// TwinCAT 3 PLC project Plc
// ProgramVersion: 3.1.4023.0
// libraries:
//   Tc2_Standard, * (Beckhoff Automation GmbH)
//   Tc2_System, * (Beckhoff Automation GmbH)
//   Tc3_Module, * (Beckhoff Automation GmbH)
// project tree:
//   / PlcTask.TcTTO (not stored)
//   DUTs/IO/PdoEntries/ FSOE_31BB7F2A.TcDUT, FSOE_3C294B21.TcDUT, FSOE_13BCEA3F.TcDUT, FSOE_6A82EB93.TcDUT, FSOE_BB3344D6.TcDUT
//   DUTs/IO/PDOs/ DeviceMain_Outputs_650F3486.TcDUT, FSoE_Slave_Connection_1_Slave_Message_330A35E4.TcDUT, Standard_Inputdata_FDD1436A.TcDUT, FSLOGIC_Inputs_CD3F9A93.TcDUT, FSoE_Slave_Connection_1_Master_Message_7109E4F0.TcDUT, Standard_Outputdata_59C030BE.TcDUT, EMPTY_STRUCTURE.TcDUT, Ch_A_AxisMain_Inputs_BA7CE8DB.TcDUT, Ch_A_AxisMain_Outputs_A99AE12E.TcDUT, Ch_A_Interpolator_Outputs_462A5F1D.TcDUT, Ch_A_PositionControl_Inputs_8CB0F55A.TcDUT, WcState_B516A264.TcDUT, InfoData_358A59CF.TcDUT, Device_6E257577.TcDUT, Device_Safety_C21945A1.TcDUT, Ch_A_D18C6F16.TcDUT, InfoData_E68C61CD.TcDUT (not stored), WcState_0B2B16F9.TcDUT (not stored), InfoData_2A97D6CF.TcDUT (not stored), Inputs_A65FACA4.TcDUT (not stored), Outputs_23C0ED1D.TcDUT (not stored)
//   DUTs/IO/Boxes/ AMP8000_F7A82895.TcDUT
//   DUTs/IO/Devices/ SyncUnitTask_2D604ED5.TcDUT (not stored), SyncUnitTasks_6FEB8257.TcDUT (not stored), SyncUnits_99E584AF.TcDUT (not stored)
//   DUTs/IO/Topology/ Device_1_EtherCAT_60A1425B.TcDUT (not stored)
//   DUTs/IO/Base/ EtcSlaveBase_82538BE2.TcDUT (not stored), EtcSlaveBase_82538BE2.TcDUT (not stored), EtcSlaveBase_82538BE2.TcDUT (not stored), EtcSlaveTerminalBase_947E5A46.TcDUT (not stored), EtcSlaveBoxBase_77A0E4A7.TcDUT (not stored), EtcSlaveEndTerminalBase_866C7F0C.TcDUT (not stored), InputBase_8311D824.TcDUT (not stored), OutputBase_10CEE7DE.TcDUT (not stored), EtcMasterBase_62654B43.TcDUT (not stored)
//   GVLs/ GVL_iXlinker.TcGVL (not stored)
// real-time tasks:
//   TASK PlcTask: cycle T#10ms, priority 20, ADS port 350
// I/O:
//   DEVICE Device 1 (EtherCAT), AmsNetId 172.20.30.238.2.1
//     Drive 1 (AMP8000-0030-0103) [AMP8000-0030-0103]
//       modules: Device, Device, Device, Device, Device, Device, Device, Device, Device, Device, Device (Safety), Device, Device, Device, Device, Device, Device, Device, Device, Device, Device, Device, Device, Device, Device, Device, Device, Device, Device, Device, Device, Ch A, Ch A, Ch A, Ch A, Ch A, Ch A, Ch A, Ch A, Ch A, Ch A, Ch A, Ch A, Ch A, Ch A, Ch A, Ch A, Ch A, Ch A, Ch A, Ch A, Ch A, Ch A, Ch A, Ch A, Ch A, Ch A
// variable links:
//   Plc/Plc Instance <-> Device 1 (EtherCAT)/Drive 1 (AMP8000-0030-0103)
//     PlcTask Outputs/GVL_iXlinker.Device_1_EtherCAT.Drive_1_AMP8000_0030_0103.Device.DeviceMain_Outputs.Power_supply_controlword <-> Device/DeviceMain Outputs/Power supply controlword
//     PlcTask Inputs/GVL_iXlinker.Device_1_EtherCAT.Drive_1_AMP8000_0030_0103.Device_Safety.FSoE_Slave_Connection_1_Slave_Message.FSOE/FSoE_Slave_Cmd <-> Device (Safety)/FSoE Slave Connection 1 Slave Message/FSOE/FSoE Slave Cmd
//     PlcTask Inputs/GVL_iXlinker.Device_1_EtherCAT.Drive_1_AMP8000_0030_0103.Device_Safety.FSoE_Slave_Connection_1_Slave_Message.FSOE/Axis_A_STO <-> Device (Safety)/FSoE Slave Connection 1 Slave Message/FSOE/Axis A STO
//     PlcTask Inputs/GVL_iXlinker.Device_1_EtherCAT.Drive_1_AMP8000_0030_0103.Device_Safety.FSoE_Slave_Connection_1_Slave_Message.FSOE/Safe_Input_1 <-> Device (Safety)/FSoE Slave Connection 1 Slave Message/FSOE/Safe Input_1
//     PlcTask Inputs/GVL_iXlinker.Device_1_EtherCAT.Drive_1_AMP8000_0030_0103.Device_Safety.FSoE_Slave_Connection_1_Slave_Message.FSOE/Safe_Input_2 <-> Device (Safety)/FSoE Slave Connection 1 Slave Message/FSOE/Safe Input_2
//     PlcTask Inputs/GVL_iXlinker.Device_1_EtherCAT.Drive_1_AMP8000_0030_0103.Device_Safety.FSoE_Slave_Connection_1_Slave_Message.FSOE/Safe_Input_3 <-> Device (Safety)/FSoE Slave Connection 1 Slave Message/FSOE/Safe Input_3
//     PlcTask Inputs/GVL_iXlinker.Device_1_EtherCAT.Drive_1_AMP8000_0030_0103.Device_Safety.FSoE_Slave_Connection_1_Slave_Message.FSOE/Safe_Input_4 <-> Device (Safety)/FSoE Slave Connection 1 Slave Message/FSOE/Safe Input_4
//     PlcTask Inputs/GVL_iXlinker.Device_1_EtherCAT.Drive_1_AMP8000_0030_0103.Device_Safety.FSoE_Slave_Connection_1_Slave_Message.FSOE/Safe_Input_5 <-> Device (Safety)/FSoE Slave Connection 1 Slave Message/FSOE/Safe Input_5
//     PlcTask Inputs/GVL_iXlinker.Device_1_EtherCAT.Drive_1_AMP8000_0030_0103.Device_Safety.FSoE_Slave_Connection_1_Slave_Message.FSOE/Safe_Input_6 <-> Device (Safety)/FSoE Slave Connection 1 Slave Message/FSOE/Safe Input_6
//     PlcTask Inputs/GVL_iXlinker.Device_1_EtherCAT.Drive_1_AMP8000_0030_0103.Device_Safety.FSoE_Slave_Connection_1_Slave_Message.FSOE/Safe_Input_7 <-> Device (Safety)/FSoE Slave Connection 1 Slave Message/FSOE/Safe Input_7
//     PlcTask Inputs/GVL_iXlinker.Device_1_EtherCAT.Drive_1_AMP8000_0030_0103.Device_Safety.FSoE_Slave_Connection_1_Slave_Message.FSOE/Safe_Input_9 <-> Device (Safety)/FSoE Slave Connection 1 Slave Message/FSOE/Safe Input_9
//     PlcTask Inputs/GVL_iXlinker.Device_1_EtherCAT.Drive_1_AMP8000_0030_0103.Device_Safety.FSoE_Slave_Connection_1_Slave_Message.FSOE/Safe_Input_10 <-> Device (Safety)/FSoE Slave Connection 1 Slave Message/FSOE/Safe Input_10
//     PlcTask Inputs/GVL_iXlinker.Device_1_EtherCAT.Drive_1_AMP8000_0030_0103.Device_Safety.FSoE_Slave_Connection_1_Slave_Message.FSOE/Safe_Input_11 <-> Device (Safety)/FSoE Slave Connection 1 Slave Message/FSOE/Safe Input_11
//     PlcTask Inputs/GVL_iXlinker.Device_1_EtherCAT.Drive_1_AMP8000_0030_0103.Device_Safety.FSoE_Slave_Connection_1_Slave_Message.FSOE/Safe_Input_12 <-> Device (Safety)/FSoE Slave Connection 1 Slave Message/FSOE/Safe Input_12
//     PlcTask Inputs/GVL_iXlinker.Device_1_EtherCAT.Drive_1_AMP8000_0030_0103.Device_Safety.FSoE_Slave_Connection_1_Slave_Message.FSOE/Safe_Input_13 <-> Device (Safety)/FSoE Slave Connection 1 Slave Message/FSOE/Safe Input_13
//     PlcTask Inputs/GVL_iXlinker.Device_1_EtherCAT.Drive_1_AMP8000_0030_0103.Device_Safety.FSoE_Slave_Connection_1_Slave_Message.FSOE/Safe_Input_14 <-> Device (Safety)/FSoE Slave Connection 1 Slave Message/FSOE/Safe Input_14
//     PlcTask Inputs/GVL_iXlinker.Device_1_EtherCAT.Drive_1_AMP8000_0030_0103.Device_Safety.FSoE_Slave_Connection_1_Slave_Message.FSOE/Safe_Input_15 <-> Device (Safety)/FSoE Slave Connection 1 Slave Message/FSOE/Safe Input_15
//     PlcTask Inputs/GVL_iXlinker.Device_1_EtherCAT.Drive_1_AMP8000_0030_0103.Device_Safety.FSoE_Slave_Connection_1_Slave_Message.FSOE/Axis_B_STO <-> Device (Safety)/FSoE Slave Connection 1 Slave Message/FSOE/Axis B STO
//     PlcTask Inputs/GVL_iXlinker.Device_1_EtherCAT.Drive_1_AMP8000_0030_0103.Device_Safety.FSoE_Slave_Connection_1_Slave_Message.FSOE/FSoE_Slave_CRC_0 <-> Device (Safety)/FSoE Slave Connection 1 Slave Message/FSOE/FSoE Slave CRC_0
//     PlcTask Inputs/GVL_iXlinker.Device_1_EtherCAT.Drive_1_AMP8000_0030_0103.Device_Safety.FSoE_Slave_Connection_1_Slave_Message.FSOE/FSoE_Slave_ConnID <-> Device (Safety)/FSoE Slave Connection 1 Slave Message/FSOE/FSoE Slave ConnID
//     PlcTask Inputs/GVL_iXlinker.Device_1_EtherCAT.Drive_1_AMP8000_0030_0103.Device_Safety.Standard_Inputdata.FSOE/Std_Input <-> Device (Safety)/Standard Inputdata/FSOE/Std Input
//     PlcTask Inputs/GVL_iXlinker.Device_1_EtherCAT.Drive_1_AMP8000_0030_0103.Device_Safety.Standard_Inputdata.FSOE/Std_Input_1 <-> Device (Safety)/Standard Inputdata/FSOE/Std Input_1
//     PlcTask Inputs/GVL_iXlinker.Device_1_EtherCAT.Drive_1_AMP8000_0030_0103.Device_Safety.Standard_Inputdata.FSOE/Std_Input_2 <-> Device (Safety)/Standard Inputdata/FSOE/Std Input_2
//     PlcTask Inputs/GVL_iXlinker.Device_1_EtherCAT.Drive_1_AMP8000_0030_0103.Device_Safety.Standard_Inputdata.FSOE/Std_Input_3 <-> Device (Safety)/Standard Inputdata/FSOE/Std Input_3
//     PlcTask Inputs/GVL_iXlinker.Device_1_EtherCAT.Drive_1_AMP8000_0030_0103.Device_Safety.Standard_Inputdata.FSOE/Std_Input_4 <-> Device (Safety)/Standard Inputdata/FSOE/Std Input_4
//     PlcTask Inputs/GVL_iXlinker.Device_1_EtherCAT.Drive_1_AMP8000_0030_0103.Device_Safety.Standard_Inputdata.FSOE/Std_Input_5 <-> Device (Safety)/Standard Inputdata/FSOE/Std Input_5
//     PlcTask Inputs/GVL_iXlinker.Device_1_EtherCAT.Drive_1_AMP8000_0030_0103.Device_Safety.Standard_Inputdata.FSOE/Std_Input_6 <-> Device (Safety)/Standard Inputdata/FSOE/Std Input_6
//     PlcTask Inputs/GVL_iXlinker.Device_1_EtherCAT.Drive_1_AMP8000_0030_0103.Device_Safety.Standard_Inputdata.FSOE/Std_Input_7 <-> Device (Safety)/Standard Inputdata/FSOE/Std Input_7
//     PlcTask Inputs/GVL_iXlinker.Device_1_EtherCAT.Drive_1_AMP8000_0030_0103.Device_Safety.FSLOGIC_Inputs.FSOE/Safe_Logic_State <-> Device (Safety)/FSLOGIC Inputs/FSOE/Safe Logic State
//     PlcTask Inputs/GVL_iXlinker.Device_1_EtherCAT.Drive_1_AMP8000_0030_0103.Device_Safety.FSLOGIC_Inputs.FSOE/Cycle_Counter <-> Device (Safety)/FSLOGIC Inputs/FSOE/Cycle Counter
//     PlcTask Outputs/GVL_iXlinker.Device_1_EtherCAT.Drive_1_AMP8000_0030_0103.Device_Safety.FSoE_Slave_Connection_1_Master_Message.FSOE/FSoE_Master_Cmd <-> Device (Safety)/FSoE Slave Connection 1 Master Message/FSOE/FSoE Master Cmd
//     PlcTask Outputs/GVL_iXlinker.Device_1_EtherCAT.Drive_1_AMP8000_0030_0103.Device_Safety.FSoE_Slave_Connection_1_Master_Message.FSOE/Axis_A_STO <-> Device (Safety)/FSoE Slave Connection 1 Master Message/FSOE/Axis A STO
//     PlcTask Outputs/GVL_iXlinker.Device_1_EtherCAT.Drive_1_AMP8000_0030_0103.Device_Safety.FSoE_Slave_Connection_1_Master_Message.FSOE/Safe_Output_1 <-> Device (Safety)/FSoE Slave Connection 1 Master Message/FSOE/Safe Output_1
//     PlcTask Outputs/GVL_iXlinker.Device_1_EtherCAT.Drive_1_AMP8000_0030_0103.Device_Safety.FSoE_Slave_Connection_1_Master_Message.FSOE/Safe_Output_2 <-> Device (Safety)/FSoE Slave Connection 1 Master Message/FSOE/Safe Output_2
//     PlcTask Outputs/GVL_iXlinker.Device_1_EtherCAT.Drive_1_AMP8000_0030_0103.Device_Safety.FSoE_Slave_Connection_1_Master_Message.FSOE/Safe_Output_3 <-> Device (Safety)/FSoE Slave Connection 1 Master Message/FSOE/Safe Output_3
//     PlcTask Outputs/GVL_iXlinker.Device_1_EtherCAT.Drive_1_AMP8000_0030_0103.Device_Safety.FSoE_Slave_Connection_1_Master_Message.FSOE/Safe_Output_4 <-> Device (Safety)/FSoE Slave Connection 1 Master Message/FSOE/Safe Output_4
//     PlcTask Outputs/GVL_iXlinker.Device_1_EtherCAT.Drive_1_AMP8000_0030_0103.Device_Safety.FSoE_Slave_Connection_1_Master_Message.FSOE/Safe_Output_5 <-> Device (Safety)/FSoE Slave Connection 1 Master Message/FSOE/Safe Output_5
//     PlcTask Outputs/GVL_iXlinker.Device_1_EtherCAT.Drive_1_AMP8000_0030_0103.Device_Safety.FSoE_Slave_Connection_1_Master_Message.FSOE/Safe_Output_6 <-> Device (Safety)/FSoE Slave Connection 1 Master Message/FSOE/Safe Output_6
//     PlcTask Outputs/GVL_iXlinker.Device_1_EtherCAT.Drive_1_AMP8000_0030_0103.Device_Safety.FSoE_Slave_Connection_1_Master_Message.FSOE/Safe_Output_7 <-> Device (Safety)/FSoE Slave Connection 1 Master Message/FSOE/Safe Output_7
//     PlcTask Outputs/GVL_iXlinker.Device_1_EtherCAT.Drive_1_AMP8000_0030_0103.Device_Safety.FSoE_Slave_Connection_1_Master_Message.FSOE/Safe_Output_9 <-> Device (Safety)/FSoE Slave Connection 1 Master Message/FSOE/Safe Output_9
//     PlcTask Outputs/GVL_iXlinker.Device_1_EtherCAT.Drive_1_AMP8000_0030_0103.Device_Safety.FSoE_Slave_Connection_1_Master_Message.FSOE/Safe_Output_10 <-> Device (Safety)/FSoE Slave Connection 1 Master Message/FSOE/Safe Output_10
//     PlcTask Outputs/GVL_iXlinker.Device_1_EtherCAT.Drive_1_AMP8000_0030_0103.Device_Safety.FSoE_Slave_Connection_1_Master_Message.FSOE/Safe_Output_11 <-> Device (Safety)/FSoE Slave Connection 1 Master Message/FSOE/Safe Output_11
//     PlcTask Outputs/GVL_iXlinker.Device_1_EtherCAT.Drive_1_AMP8000_0030_0103.Device_Safety.FSoE_Slave_Connection_1_Master_Message.FSOE/Safe_Output_12 <-> Device (Safety)/FSoE Slave Connection 1 Master Message/FSOE/Safe Output_12
//     PlcTask Outputs/GVL_iXlinker.Device_1_EtherCAT.Drive_1_AMP8000_0030_0103.Device_Safety.FSoE_Slave_Connection_1_Master_Message.FSOE/Safe_Output_13 <-> Device (Safety)/FSoE Slave Connection 1 Master Message/FSOE/Safe Output_13
//     PlcTask Outputs/GVL_iXlinker.Device_1_EtherCAT.Drive_1_AMP8000_0030_0103.Device_Safety.FSoE_Slave_Connection_1_Master_Message.FSOE/Safe_Output_14 <-> Device (Safety)/FSoE Slave Connection 1 Master Message/FSOE/Safe Output_14
//     PlcTask Outputs/GVL_iXlinker.Device_1_EtherCAT.Drive_1_AMP8000_0030_0103.Device_Safety.FSoE_Slave_Connection_1_Master_Message.FSOE/Safe_Output_15 <-> Device (Safety)/FSoE Slave Connection 1 Master Message/FSOE/Safe Output_15
//     PlcTask Outputs/GVL_iXlinker.Device_1_EtherCAT.Drive_1_AMP8000_0030_0103.Device_Safety.FSoE_Slave_Connection_1_Master_Message.FSOE/Axis_B_STO <-> Device (Safety)/FSoE Slave Connection 1 Master Message/FSOE/Axis B STO
//     PlcTask Outputs/GVL_iXlinker.Device_1_EtherCAT.Drive_1_AMP8000_0030_0103.Device_Safety.FSoE_Slave_Connection_1_Master_Message.FSOE/FSoE_Master_CRC_0 <-> Device (Safety)/FSoE Slave Connection 1 Master Message/FSOE/FSoE Master CRC_0
//     PlcTask Outputs/GVL_iXlinker.Device_1_EtherCAT.Drive_1_AMP8000_0030_0103.Device_Safety.FSoE_Slave_Connection_1_Master_Message.FSOE/FSoE_Master_ConnID <-> Device (Safety)/FSoE Slave Connection 1 Master Message/FSOE/FSoE Master ConnID
//     PlcTask Outputs/GVL_iXlinker.Device_1_EtherCAT.Drive_1_AMP8000_0030_0103.Device_Safety.Standard_Outputdata.FSOE/Std_Output <-> Device (Safety)/Standard Outputdata/FSOE/Std Output
//     PlcTask Outputs/GVL_iXlinker.Device_1_EtherCAT.Drive_1_AMP8000_0030_0103.Device_Safety.Standard_Outputdata.FSOE/Std_Output_1 <-> Device (Safety)/Standard Outputdata/FSOE/Std Output_1
//     PlcTask Outputs/GVL_iXlinker.Device_1_EtherCAT.Drive_1_AMP8000_0030_0103.Device_Safety.Standard_Outputdata.FSOE/Std_Output_2 <-> Device (Safety)/Standard Outputdata/FSOE/Std Output_2
//     PlcTask Outputs/GVL_iXlinker.Device_1_EtherCAT.Drive_1_AMP8000_0030_0103.Device_Safety.Standard_Outputdata.FSOE/Std_Output_3 <-> Device (Safety)/Standard Outputdata/FSOE/Std Output_3
//     PlcTask Outputs/GVL_iXlinker.Device_1_EtherCAT.Drive_1_AMP8000_0030_0103.Device_Safety.Standard_Outputdata.FSOE/Std_Output_4 <-> Device (Safety)/Standard Outputdata/FSOE/Std Output_4
//     PlcTask Outputs/GVL_iXlinker.Device_1_EtherCAT.Drive_1_AMP8000_0030_0103.Device_Safety.Standard_Outputdata.FSOE/Std_Output_5 <-> Device (Safety)/Standard Outputdata/FSOE/Std Output_5
//     PlcTask Outputs/GVL_iXlinker.Device_1_EtherCAT.Drive_1_AMP8000_0030_0103.Device_Safety.Standard_Outputdata.FSOE/Std_Output_6 <-> Device (Safety)/Standard Outputdata/FSOE/Std Output_6
//     PlcTask Outputs/GVL_iXlinker.Device_1_EtherCAT.Drive_1_AMP8000_0030_0103.Device_Safety.Standard_Outputdata.FSOE/Std_Output_7 <-> Device (Safety)/Standard Outputdata/FSOE/Std Output_7
//     PlcTask Inputs/GVL_iXlinker.Device_1_EtherCAT.Drive_1_AMP8000_0030_0103.Ch_A.Ch_A_AxisMain_Inputs.Position_actual_value_invalid <-> Ch A/Ch A AxisMain Inputs/Position actual value invalid
//     PlcTask Inputs/GVL_iXlinker.Device_1_EtherCAT.Drive_1_AMP8000_0030_0103.Ch_A.Ch_A_AxisMain_Inputs._1st_Additional_position_actual_value_invalid <-> Ch A/Ch A AxisMain Inputs/1st Additional position actual value invalid
//     PlcTask Inputs/GVL_iXlinker.Device_1_EtherCAT.Drive_1_AMP8000_0030_0103.Ch_A.Ch_A_AxisMain_Inputs.Ch_A_Statusword <-> Ch A/Ch A AxisMain Inputs/Ch A Statusword
//     PlcTask Inputs/GVL_iXlinker.Device_1_EtherCAT.Drive_1_AMP8000_0030_0103.Ch_A.Ch_A_AxisMain_Inputs.Ch_A_Position_actual_value <-> Ch A/Ch A AxisMain Inputs/Ch A Position actual value
//     PlcTask Outputs/GVL_iXlinker.Device_1_EtherCAT.Drive_1_AMP8000_0030_0103.Ch_A.Ch_A_AxisMain_Outputs.Ch_A_Controlword <-> Ch A/Ch A AxisMain Outputs/Ch A Controlword
//     PlcTask Outputs/GVL_iXlinker.Device_1_EtherCAT.Drive_1_AMP8000_0030_0103.Ch_A.Ch_A_Interpolator_Outputs.Ch_A_Target_position <-> Ch A/Ch A Interpolator Outputs/Ch A Target position
//     PlcTask Outputs/GVL_iXlinker.Device_1_EtherCAT.Drive_1_AMP8000_0030_0103.Ch_A.Ch_A_Interpolator_Outputs.Ch_A_Target_velocity <-> Ch A/Ch A Interpolator Outputs/Ch A Target velocity
//     PlcTask Inputs/GVL_iXlinker.Device_1_EtherCAT.Drive_1_AMP8000_0030_0103.Ch_A.Ch_A_PositionControl_Inputs.Ch_A_Following_error_actual_value <-> Ch A/Ch A PositionControl Inputs/Ch A Following error actual value
//     PlcTask Inputs/GVL_iXlinker.Device_1_EtherCAT.Drive_1_AMP8000_0030_0103.WcState.WcState0 <-> WcState/WcState0
//     PlcTask Inputs/GVL_iXlinker.Device_1_EtherCAT.Drive_1_AMP8000_0030_0103.WcState.WcState1 <-> WcState/WcState1
//     PlcTask Inputs/GVL_iXlinker.Device_1_EtherCAT.Drive_1_AMP8000_0030_0103.WcState.InputToggle0 <-> WcState/InputToggle0
//     PlcTask Inputs/GVL_iXlinker.Device_1_EtherCAT.Drive_1_AMP8000_0030_0103.WcState.InputToggle1 <-> WcState/InputToggle1
//     PlcTask Inputs/GVL_iXlinker.Device_1_EtherCAT.Drive_1_AMP8000_0030_0103.InfoData.AdsAddr <-> InfoData/AdsAddr
//     PlcTask Inputs/GVL_iXlinker.Device_1_EtherCAT.Drive_1_AMP8000_0030_0103.InfoData.DcOutputShift <-> InfoData/DcOutputShift
//     PlcTask Inputs/GVL_iXlinker.Device_1_EtherCAT.Drive_1_AMP8000_0030_0103.InfoData.DcInputShift <-> InfoData/DcInputShift
//     PlcTask Inputs/GVL_iXlinker.Device_1_EtherCAT.Drive_1_AMP8000_0030_0103.InfoData.AoeNetId <-> InfoData/AoeNetId
//     PlcTask Inputs/GVL_iXlinker.Device_1_EtherCAT.Drive_1_AMP8000_0030_0103.InfoData.Chn0 <-> InfoData/Chn0
//     PlcTask Inputs/GVL_iXlinker.Device_1_EtherCAT.Drive_1_AMP8000_0030_0103.InfoData.State <-> InfoData/State
//   Plc/Plc Instance <-> Device 1 (EtherCAT)
//     PlcTask Inputs/GVL_iXlinker.Device_1_EtherCAT.SyncUnits._default._unreferenced.WcState.WcState <-> SyncUnits/<default>/<unreferenced>/WcState/WcState
//     PlcTask Inputs/GVL_iXlinker.Device_1_EtherCAT.SyncUnits._default._unreferenced.InfoData.ObjectId <-> SyncUnits/<default>/<unreferenced>/InfoData/ObjectId
//     PlcTask Inputs/GVL_iXlinker.Device_1_EtherCAT.SyncUnits._default._unreferenced.InfoData.State <-> SyncUnits/<default>/<unreferenced>/InfoData/State
//     PlcTask Inputs/GVL_iXlinker.Device_1_EtherCAT.SyncUnits._default._unreferenced.InfoData.SlaveCount <-> SyncUnits/<default>/<unreferenced>/InfoData/SlaveCount
//     PlcTask Inputs/GVL_iXlinker.Device_1_EtherCAT.SyncUnits._default.PlcTask.WcState.WcState <-> SyncUnits/<default>/PlcTask/WcState/WcState
//     PlcTask Inputs/GVL_iXlinker.Device_1_EtherCAT.SyncUnits._default.PlcTask.InfoData.ObjectId <-> SyncUnits/<default>/PlcTask/InfoData/ObjectId
//     PlcTask Inputs/GVL_iXlinker.Device_1_EtherCAT.SyncUnits._default.PlcTask.InfoData.State <-> SyncUnits/<default>/PlcTask/InfoData/State
//     PlcTask Inputs/GVL_iXlinker.Device_1_EtherCAT.SyncUnits._default.PlcTask.InfoData.SlaveCount <-> SyncUnits/<default>/PlcTask/InfoData/SlaveCount
//     PlcTask Inputs/GVL_iXlinker.Device_1_EtherCAT.Inputs.SlaveCount <-> Inputs/SlaveCount
//     PlcTask Inputs/GVL_iXlinker.Device_1_EtherCAT.Inputs.DevState <-> Inputs/DevState
//     PlcTask Inputs/GVL_iXlinker.Device_1_EtherCAT.Inputs.Frm0State <-> Inputs/Frm0State
//     PlcTask Inputs/GVL_iXlinker.Device_1_EtherCAT.Inputs.Frm0WcState <-> Inputs/Frm0WcState
//     PlcTask Inputs/GVL_iXlinker.Device_1_EtherCAT.Inputs.Frm0InputToggle <-> Inputs/Frm0InputToggle
//     PlcTask Outputs/GVL_iXlinker.Device_1_EtherCAT.Outputs.DevCtrl <-> Outputs/DevCtrl
//     PlcTask Outputs/GVL_iXlinker.Device_1_EtherCAT.Outputs.Frm0Ctrl <-> Outputs/Frm0Ctrl
//     PlcTask Outputs/GVL_iXlinker.Device_1_EtherCAT.Outputs.Frm0WcCtrl <-> Outputs/Frm0WcCtrl
//     PlcTask Inputs/GVL_iXlinker.Device_1_EtherCAT.InfoData.ChangeCount <-> InfoData/ChangeCount
//     PlcTask Inputs/GVL_iXlinker.Device_1_EtherCAT.InfoData.DevId <-> InfoData/DevId
//     PlcTask Inputs/GVL_iXlinker.Device_1_EtherCAT.InfoData.AmsNetId <-> InfoData/AmsNetId
//     PlcTask Inputs/GVL_iXlinker.Device_1_EtherCAT.InfoData.CfgSlaveCount <-> InfoData/CfgSlaveCount
//     PlcTask Inputs/GVL_iXlinker.Device_1_EtherCAT.InfoData.DcToTcTimeOffset <-> InfoData/DcToTcTimeOffset
//     PlcTask Inputs/GVL_iXlinker.Device_1_EtherCAT.InfoData.DcToExtTimeOffset <-> InfoData/DcToExtTimeOffset

// ---- DUTs/IO/PdoEntries/FSOE_31BB7F2A.TcDUT
{attribute 'GeneratedUsingTerminal: AMP8000-0030-0103-0103'}
{attribute addProperty BoxType "AMP8000-0030-0103-0103"}
{attribute addProperty Id "FSoE_Slave_CmdUSINT1Axis_A_STOBOOL1Safe_Input_1BOOL1Safe_Input_2BOOL1Safe_Input_3BOOL1Safe_Input_4BOOL1Safe_Input_5BOOL1Safe_Input_6BOOL1Safe_Input_7BOOL1Axis_B_STOBOOL1Safe_Input_9BOOL1Safe_Input_10BOOL1Safe_Input_11BOOL1Safe_Input_12BOOL1Safe_Input_13BOOL1Safe_Input_14BOOL1Safe_Input_15BOOL1FSoE_Slave_CRC_0UINT2FSoE_Slave_ConnIDUINT2"}
{attribute addProperty CRC "834371370"}
{attribute addProperty Size "21"}
TYPE FSOE_31BB7F2A :
STRUCT
	{attribute addProperty Name "FSoE_Slave_Cmd"}
	FSoE_Slave_Cmd : USINT;
	{attribute addProperty Name "Axis_A_STO"}
	Axis_A_STO : BOOL;
	{attribute addProperty Name "Safe_Input_1"}
	Safe_Input_1 : BOOL;
	{attribute addProperty Name "Safe_Input_2"}
	Safe_Input_2 : BOOL;
	{attribute addProperty Name "Safe_Input_3"}
	Safe_Input_3 : BOOL;
	{attribute addProperty Name "Safe_Input_4"}
	Safe_Input_4 : BOOL;
	{attribute addProperty Name "Safe_Input_5"}
	Safe_Input_5 : BOOL;
	{attribute addProperty Name "Safe_Input_6"}
	Safe_Input_6 : BOOL;
	{attribute addProperty Name "Safe_Input_7"}
	Safe_Input_7 : BOOL;
	{attribute addProperty Name "Axis_B_STO"}
	Axis_B_STO : BOOL;
	{attribute addProperty Name "Safe_Input_9"}
	Safe_Input_9 : BOOL;
	{attribute addProperty Name "Safe_Input_10"}
	Safe_Input_10 : BOOL;
	{attribute addProperty Name "Safe_Input_11"}
	Safe_Input_11 : BOOL;
	{attribute addProperty Name "Safe_Input_12"}
	Safe_Input_12 : BOOL;
	{attribute addProperty Name "Safe_Input_13"}
	Safe_Input_13 : BOOL;
	{attribute addProperty Name "Safe_Input_14"}
	Safe_Input_14 : BOOL;
	{attribute addProperty Name "Safe_Input_15"}
	Safe_Input_15 : BOOL;
	{attribute addProperty Name "FSoE_Slave_CRC_0"}
	FSoE_Slave_CRC_0 : UINT;
	{attribute addProperty Name "FSoE_Slave_ConnID"}
	FSoE_Slave_ConnID : UINT;
END_STRUCT
END_TYPE

// ---- DUTs/IO/PdoEntries/FSOE_3C294B21.TcDUT
{attribute 'GeneratedUsingTerminal: AMP8000-0030-0103-0103'}
{attribute addProperty BoxType "AMP8000-0030-0103-0103"}
{attribute addProperty Id "Std_InputBOOL1Std_Input_1BOOL1Std_Input_2BOOL1Std_Input_3BOOL1Std_Input_4BOOL1Std_Input_5BOOL1Std_Input_6BOOL1Std_Input_7BOOL1"}
{attribute addProperty CRC "1009339169"}
{attribute addProperty Size "8"}
TYPE FSOE_3C294B21 :
STRUCT
	{attribute addProperty Name "Std_Input"}
	Std_Input : BOOL;
	{attribute addProperty Name "Std_Input_1"}
	Std_Input_1 : BOOL;
	{attribute addProperty Name "Std_Input_2"}
	Std_Input_2 : BOOL;
	{attribute addProperty Name "Std_Input_3"}
	Std_Input_3 : BOOL;
	{attribute addProperty Name "Std_Input_4"}
	Std_Input_4 : BOOL;
	{attribute addProperty Name "Std_Input_5"}
	Std_Input_5 : BOOL;
	{attribute addProperty Name "Std_Input_6"}
	Std_Input_6 : BOOL;
	{attribute addProperty Name "Std_Input_7"}
	Std_Input_7 : BOOL;
END_STRUCT
END_TYPE

// ---- DUTs/IO/PdoEntries/FSOE_13BCEA3F.TcDUT
{attribute 'GeneratedUsingTerminal: AMP8000-0030-0103-0103'}
{attribute addProperty BoxType "AMP8000-0030-0103-0103"}
{attribute addProperty Id "Safe_Logic_StateUSINT1Cycle_CounterUSINT1"}
{attribute addProperty CRC "331147839"}
{attribute addProperty Size "2"}
TYPE FSOE_13BCEA3F :
STRUCT
	{attribute addProperty Name "Safe_Logic_State"}
	Safe_Logic_State : USINT;
	{attribute addProperty Name "Cycle_Counter"}
	Cycle_Counter : USINT;
END_STRUCT
END_TYPE

// ---- DUTs/IO/PdoEntries/FSOE_6A82EB93.TcDUT
{attribute 'GeneratedUsingTerminal: AMP8000-0030-0103-0103'}
{attribute addProperty BoxType "AMP8000-0030-0103-0103"}
{attribute addProperty Id "FSoE_Master_CmdUSINT1Axis_A_STOBOOL1Safe_Output_1BOOL1Safe_Output_2BOOL1Safe_Output_3BOOL1Safe_Output_4BOOL1Safe_Output_5BOOL1Safe_Output_6BOOL1Safe_Output_7BOOL1Axis_B_STOBOOL1Safe_Output_9BOOL1Safe_Output_10BOOL1Safe_Output_11BOOL1Safe_Output_12BOOL1Safe_Output_13BOOL1Safe_Output_14BOOL1Safe_Output_15BOOL1FSoE_Master_CRC_0UINT2FSoE_Master_ConnIDUINT2"}
{attribute addProperty CRC "1786964883"}
{attribute addProperty Size "21"}
TYPE FSOE_6A82EB93 :
STRUCT
	{attribute addProperty Name "FSoE_Master_Cmd"}
	FSoE_Master_Cmd : USINT;
	{attribute addProperty Name "Axis_A_STO"}
	Axis_A_STO : BOOL;
	{attribute addProperty Name "Safe_Output_1"}
	Safe_Output_1 : BOOL;
	{attribute addProperty Name "Safe_Output_2"}
	Safe_Output_2 : BOOL;
	{attribute addProperty Name "Safe_Output_3"}
	Safe_Output_3 : BOOL;
	{attribute addProperty Name "Safe_Output_4"}
	Safe_Output_4 : BOOL;
	{attribute addProperty Name "Safe_Output_5"}
	Safe_Output_5 : BOOL;
	{attribute addProperty Name "Safe_Output_6"}
	Safe_Output_6 : BOOL;
	{attribute addProperty Name "Safe_Output_7"}
	Safe_Output_7 : BOOL;
	{attribute addProperty Name "Axis_B_STO"}
	Axis_B_STO : BOOL;
	{attribute addProperty Name "Safe_Output_9"}
	Safe_Output_9 : BOOL;
	{attribute addProperty Name "Safe_Output_10"}
	Safe_Output_10 : BOOL;
	{attribute addProperty Name "Safe_Output_11"}
	Safe_Output_11 : BOOL;
	{attribute addProperty Name "Safe_Output_12"}
	Safe_Output_12 : BOOL;
	{attribute addProperty Name "Safe_Output_13"}
	Safe_Output_13 : BOOL;
	{attribute addProperty Name "Safe_Output_14"}
	Safe_Output_14 : BOOL;
	{attribute addProperty Name "Safe_Output_15"}
	Safe_Output_15 : BOOL;
	{attribute addProperty Name "FSoE_Master_CRC_0"}
	FSoE_Master_CRC_0 : UINT;
	{attribute addProperty Name "FSoE_Master_ConnID"}
	FSoE_Master_ConnID : UINT;
END_STRUCT
END_TYPE

// ---- DUTs/IO/PdoEntries/FSOE_BB3344D6.TcDUT
{attribute 'GeneratedUsingTerminal: AMP8000-0030-0103-0103'}
{attribute addProperty BoxType "AMP8000-0030-0103-0103"}
{attribute addProperty Id "Std_OutputBOOL1Std_Output_1BOOL1Std_Output_2BOOL1Std_Output_3BOOL1Std_Output_4BOOL1Std_Output_5BOOL1Std_Output_6BOOL1Std_Output_7BOOL1"}
{attribute addProperty CRC "3140699350"}
{attribute addProperty Size "8"}
TYPE FSOE_BB3344D6 :
STRUCT
	{attribute addProperty Name "Std_Output"}
	Std_Output : BOOL;
	{attribute addProperty Name "Std_Output_1"}
	Std_Output_1 : BOOL;
	{attribute addProperty Name "Std_Output_2"}
	Std_Output_2 : BOOL;
	{attribute addProperty Name "Std_Output_3"}
	Std_Output_3 : BOOL;
	{attribute addProperty Name "Std_Output_4"}
	Std_Output_4 : BOOL;
	{attribute addProperty Name "Std_Output_5"}
	Std_Output_5 : BOOL;
	{attribute addProperty Name "Std_Output_6"}
	Std_Output_6 : BOOL;
	{attribute addProperty Name "Std_Output_7"}
	Std_Output_7 : BOOL;
END_STRUCT
END_TYPE

// ---- DUTs/IO/PDOs/DeviceMain_Outputs_650F3486.TcDUT
{attribute 'GeneratedUsingTerminal: AMP8000-0030-0103-0103'}
{attribute addProperty BoxType "AMP8000-0030-0103-0103"}
{attribute addProperty Id "Power_supply_controlwordAT %Q*UINT2"}
{attribute addProperty CRC "1695495302"}
{attribute addProperty Size "2"}
TYPE DeviceMain_Outputs_650F3486 EXTENDS OutputBase_10CEE7DE :
STRUCT
	{attribute addProperty Name "Power_supply_controlword"}
	Power_supply_controlword AT %Q* : UINT;
END_STRUCT
END_TYPE

// ---- DUTs/IO/PDOs/FSoE_Slave_Connection_1_Slave_Message_330A35E4.TcDUT
{attribute 'GeneratedUsingTerminal: AMP8000-0030-0103-0103'}
{attribute addProperty BoxType "AMP8000-0030-0103-0103"}
{attribute addProperty Id "FSOEAT %I*FSOE_31BB7F2A21"}
{attribute addProperty CRC "856307172"}
{attribute addProperty Size "21"}
TYPE FSoE_Slave_Connection_1_Slave_Message_330A35E4 EXTENDS InputBase_8311D824 :
STRUCT
	{attribute addProperty Name "FSOE"}
	FSOE AT %I* : FSOE_31BB7F2A;
END_STRUCT
END_TYPE

// ---- DUTs/IO/PDOs/Standard_Inputdata_FDD1436A.TcDUT
{attribute 'GeneratedUsingTerminal: AMP8000-0030-0103-0103'}
{attribute addProperty BoxType "AMP8000-0030-0103-0103"}
{attribute addProperty Id "FSOEAT %I*FSOE_3C294B218"}
{attribute addProperty CRC "4258349930"}
{attribute addProperty Size "8"}
TYPE Standard_Inputdata_FDD1436A EXTENDS InputBase_8311D824 :
STRUCT
	{attribute addProperty Name "FSOE"}
	FSOE AT %I* : FSOE_3C294B21;
END_STRUCT
END_TYPE

// ---- DUTs/IO/PDOs/FSLOGIC_Inputs_CD3F9A93.TcDUT
{attribute 'GeneratedUsingTerminal: AMP8000-0030-0103-0103'}
{attribute addProperty BoxType "AMP8000-0030-0103-0103"}
{attribute addProperty Id "FSOEAT %I*FSOE_13BCEA3F2"}
{attribute addProperty CRC "3443497619"}
{attribute addProperty Size "2"}
TYPE FSLOGIC_Inputs_CD3F9A93 EXTENDS InputBase_8311D824 :
STRUCT
	{attribute addProperty Name "FSOE"}
	FSOE AT %I* : FSOE_13BCEA3F;
END_STRUCT
END_TYPE

// ---- DUTs/IO/PDOs/FSoE_Slave_Connection_1_Master_Message_7109E4F0.TcDUT
{attribute 'GeneratedUsingTerminal: AMP8000-0030-0103-0103'}
{attribute addProperty BoxType "AMP8000-0030-0103-0103"}
{attribute addProperty Id "FSOEAT %Q*FSOE_6A82EB9321"}
{attribute addProperty CRC "1896473840"}
{attribute addProperty Size "21"}
TYPE FSoE_Slave_Connection_1_Master_Message_7109E4F0 EXTENDS OutputBase_10CEE7DE :
STRUCT
	{attribute addProperty Name "FSOE"}
	FSOE AT %Q* : FSOE_6A82EB93;
END_STRUCT
END_TYPE

// ---- DUTs/IO/PDOs/Standard_Outputdata_59C030BE.TcDUT
{attribute 'GeneratedUsingTerminal: AMP8000-0030-0103-0103'}
{attribute addProperty BoxType "AMP8000-0030-0103-0103"}
{attribute addProperty Id "FSOEAT %Q*FSOE_BB3344D68"}
{attribute addProperty CRC "1505767614"}
{attribute addProperty Size "8"}
TYPE Standard_Outputdata_59C030BE EXTENDS OutputBase_10CEE7DE :
STRUCT
	{attribute addProperty Name "FSOE"}
	FSOE AT %Q* : FSOE_BB3344D6;
END_STRUCT
END_TYPE

// ---- DUTs/IO/PDOs/EMPTY_STRUCTURE.TcDUT
{attribute 'GeneratedUsingTerminal: AMP8000-0030-0103-0103'}
{attribute addProperty BoxType "AMP8000-0030-0103-0103"}
{attribute addProperty Id "EMPTY_STRUCTURE"}
{attribute addProperty CRC "0"}
{attribute addProperty Size "0"}
TYPE EMPTY_STRUCTURE :
STRUCT
END_STRUCT
END_TYPE

// ---- DUTs/IO/PDOs/Ch_A_AxisMain_Inputs_BA7CE8DB.TcDUT
{attribute 'GeneratedUsingTerminal: AMP8000-0030-0103-0103'}
{attribute addProperty BoxType "AMP8000-0030-0103-0103"}
{attribute addProperty Id "Position_actual_value_invalidAT %I*BOOL1_1st_Additional_position_actual_value_invalidAT %I*BOOL1Ch_A_StatuswordAT %I*UINT2Ch_A_Position_actual_valueAT %I*DINT4"}
{attribute addProperty CRC "3128748251"}
{attribute addProperty Size "8"}
TYPE Ch_A_AxisMain_Inputs_BA7CE8DB EXTENDS InputBase_8311D824 :
STRUCT
	{attribute addProperty Name "Position_actual_value_invalid"}
	Position_actual_value_invalid AT %I* : BOOL;
	{attribute addProperty Name "_1st_Additional_position_actual_value_invalid"}
	_1st_Additional_position_actual_value_invalid AT %I* : BOOL;
	{attribute addProperty Name "Ch_A_Statusword"}
	Ch_A_Statusword AT %I* : UINT;
	{attribute addProperty Name "Ch_A_Position_actual_value"}
	Ch_A_Position_actual_value AT %I* : DINT;
END_STRUCT
END_TYPE

// ---- DUTs/IO/PDOs/Ch_A_AxisMain_Outputs_A99AE12E.TcDUT
{attribute 'GeneratedUsingTerminal: AMP8000-0030-0103-0103'}
{attribute addProperty BoxType "AMP8000-0030-0103-0103"}
{attribute addProperty Id "Ch_A_ControlwordAT %Q*UINT2"}
{attribute addProperty CRC "2845499694"}
{attribute addProperty Size "2"}
TYPE Ch_A_AxisMain_Outputs_A99AE12E EXTENDS OutputBase_10CEE7DE :
STRUCT
	{attribute addProperty Name "Ch_A_Controlword"}
	Ch_A_Controlword AT %Q* : UINT;
END_STRUCT
END_TYPE

// ---- DUTs/IO/PDOs/Ch_A_Interpolator_Outputs_462A5F1D.TcDUT
{attribute 'GeneratedUsingTerminal: AMP8000-0030-0103-0103'}
{attribute addProperty BoxType "AMP8000-0030-0103-0103"}
{attribute addProperty Id "Ch_A_Target_positionAT %Q*DINT4Ch_A_Target_velocityAT %Q*DINT4"}
{attribute addProperty CRC "1177181981"}
{attribute addProperty Size "8"}
TYPE Ch_A_Interpolator_Outputs_462A5F1D EXTENDS OutputBase_10CEE7DE :
STRUCT
	{attribute addProperty Name "Ch_A_Target_position"}
	Ch_A_Target_position AT %Q* : DINT;
	{attribute addProperty Name "Ch_A_Target_velocity"}
	Ch_A_Target_velocity AT %Q* : DINT;
END_STRUCT
END_TYPE

// ---- DUTs/IO/PDOs/Ch_A_PositionControl_Inputs_8CB0F55A.TcDUT
{attribute 'GeneratedUsingTerminal: AMP8000-0030-0103-0103'}
{attribute addProperty BoxType "AMP8000-0030-0103-0103"}
{attribute addProperty Id "Ch_A_Following_error_actual_valueAT %I*DINT4"}
{attribute addProperty CRC "2360407386"}
{attribute addProperty Size "4"}
TYPE Ch_A_PositionControl_Inputs_8CB0F55A EXTENDS InputBase_8311D824 :
STRUCT
	{attribute addProperty Name "Ch_A_Following_error_actual_value"}
	Ch_A_Following_error_actual_value AT %I* : DINT;
END_STRUCT
END_TYPE

// ---- DUTs/IO/PDOs/WcState_B516A264.TcDUT
{attribute 'GeneratedUsingTerminal: AMP8000-0030-0103-0103'}
{attribute addProperty BoxType "AMP8000-0030-0103-0103"}
{attribute addProperty Id "WcState0AT %I*BOOL1WcState1AT %I*BOOL1InputToggle0AT %I*BOOL1InputToggle1AT %I*BOOL1"}
{attribute addProperty CRC "3038159460"}
{attribute addProperty Size "4"}
TYPE WcState_B516A264 EXTENDS InputBase_8311D824 :
STRUCT
	{attribute addProperty Name "WcState0"}
	WcState0 AT %I* : BOOL;
	{attribute addProperty Name "WcState1"}
	WcState1 AT %I* : BOOL;
	{attribute addProperty Name "InputToggle0"}
	InputToggle0 AT %I* : BOOL;
	{attribute addProperty Name "InputToggle1"}
	InputToggle1 AT %I* : BOOL;
END_STRUCT
END_TYPE

// ---- DUTs/IO/PDOs/InfoData_358A59CF.TcDUT
{attribute 'GeneratedUsingTerminal: AMP8000-0030-0103-0103'}
{attribute addProperty BoxType "AMP8000-0030-0103-0103"}
{attribute addProperty Id "AdsAddrAT %I*AMSADDR8DcOutputShiftAT %I*DINT4DcInputShiftAT %I*DINT4AoeNetIdAT %I*AMSNETID6Chn0AT %I*USINT1StateAT %I*UINT2"}
{attribute addProperty CRC "898259407"}
{attribute addProperty Size "25"}
TYPE InfoData_358A59CF EXTENDS InputBase_8311D824 :
STRUCT
	{attribute addProperty Name "AdsAddr"}
	AdsAddr AT %I* : AMSADDR;
	{attribute addProperty Name "DcOutputShift"}
	DcOutputShift AT %I* : DINT;
	{attribute addProperty Name "DcInputShift"}
	DcInputShift AT %I* : DINT;
	{attribute addProperty Name "AoeNetId"}
	AoeNetId AT %I* : AMSNETID;
	{attribute addProperty Name "Chn0"}
	Chn0 AT %I* : USINT;
	{attribute addProperty Name "State"}
	State AT %I* : UINT;
END_STRUCT
END_TYPE

// ---- DUTs/IO/PDOs/Device_6E257577.TcDUT
{attribute 'GeneratedUsingTerminal: AMP8000-0030-0103-0103'}
{attribute addProperty BoxType "AMP8000-0030-0103-0103"}
{attribute addProperty Id "DeviceMain_OutputsDeviceMain_Outputs_650F34862"}
{attribute addProperty CRC "1847948663"}
{attribute addProperty Size "2"}
TYPE Device_6E257577 :
STRUCT
	{attribute addProperty Name "DeviceMain_Outputs"}
	DeviceMain_Outputs  : DeviceMain_Outputs_650F3486;
END_STRUCT
END_TYPE

// ---- DUTs/IO/PDOs/Device_Safety_C21945A1.TcDUT
{attribute 'GeneratedUsingTerminal: AMP8000-0030-0103-0103'}
{attribute addProperty BoxType "AMP8000-0030-0103-0103"}
{attribute addProperty Id "FSoE_Slave_Connection_1_Slave_MessageFSoE_Slave_Connection_1_Slave_Message_330A35E421Standard_InputdataStandard_Inputdata_FDD1436A8FSLOGIC_InputsFSLOGIC_Inputs_CD3F9A932FSoE_Slave_Connection_1_Master_MessageFSoE_Slave_Connection_1_Master_Message_7109E4F021Standard_OutputdataStandard_Outputdata_59C030BE8FSLOGIC_OutputsEMPTY_STRUCTURE0"}
{attribute addProperty CRC "3256436129"}
{attribute addProperty Size "60"}
TYPE Device_Safety_C21945A1 :
STRUCT
	{attribute addProperty Name "FSoE_Slave_Connection_1_Slave_Message"}
	FSoE_Slave_Connection_1_Slave_Message  : FSoE_Slave_Connection_1_Slave_Message_330A35E4;
	{attribute addProperty Name "Standard_Inputdata"}
	Standard_Inputdata  : Standard_Inputdata_FDD1436A;
	{attribute addProperty Name "FSLOGIC_Inputs"}
	FSLOGIC_Inputs  : FSLOGIC_Inputs_CD3F9A93;
	{attribute addProperty Name "FSoE_Slave_Connection_1_Master_Message"}
	FSoE_Slave_Connection_1_Master_Message  : FSoE_Slave_Connection_1_Master_Message_7109E4F0;
	{attribute addProperty Name "Standard_Outputdata"}
	Standard_Outputdata  : Standard_Outputdata_59C030BE;
	{attribute addProperty Name "FSLOGIC_Outputs"}
	FSLOGIC_Outputs  : EMPTY_STRUCTURE;
END_STRUCT
END_TYPE

// ---- DUTs/IO/PDOs/Ch_A_D18C6F16.TcDUT
{attribute 'GeneratedUsingTerminal: AMP8000-0030-0103-0103'}
{attribute addProperty BoxType "AMP8000-0030-0103-0103"}
{attribute addProperty Id "Ch_A_AxisMain_InputsCh_A_AxisMain_Inputs_BA7CE8DB8Ch_A_AxisMain_OutputsCh_A_AxisMain_Outputs_A99AE12E2Ch_A_Interpolator_OutputsCh_A_Interpolator_Outputs_462A5F1D8Ch_A_PositionControl_InputsCh_A_PositionControl_Inputs_8CB0F55A4"}
{attribute addProperty CRC "3515641622"}
{attribute addProperty Size "22"}
TYPE Ch_A_D18C6F16 :
STRUCT
	{attribute addProperty Name "Ch_A_AxisMain_Inputs"}
	Ch_A_AxisMain_Inputs  : Ch_A_AxisMain_Inputs_BA7CE8DB;
	{attribute addProperty Name "Ch_A_AxisMain_Outputs"}
	Ch_A_AxisMain_Outputs  : Ch_A_AxisMain_Outputs_A99AE12E;
	{attribute addProperty Name "Ch_A_Interpolator_Outputs"}
	Ch_A_Interpolator_Outputs  : Ch_A_Interpolator_Outputs_462A5F1D;
	{attribute addProperty Name "Ch_A_PositionControl_Inputs"}
	Ch_A_PositionControl_Inputs  : Ch_A_PositionControl_Inputs_8CB0F55A;
END_STRUCT
END_TYPE

// ---- DUTs/IO/Boxes/AMP8000_F7A82895.TcDUT
{attribute 'GeneratedUsingTerminal: AMP8000-0030-0103-0103'}
{attribute addProperty BoxType "AMP8000-0030-0103-0103"}
{attribute addProperty Description "AMP8000-0030-0103"}
{attribute addProperty Physics "Y"}
{attribute addProperty Id "DeviceDevice_6E2575772Device_SafetyDevice_Safety_C21945A160Ch_ACh_A_D18C6F1622WcStateAT %I*WcState_B516A2644InfoDataAT %I*InfoData_358A59CF25"}
{attribute addProperty CRC "4154992789"}
{attribute addProperty Size "113"}
TYPE AMP8000_F7A82895 EXTENDS EtcSlaveBoxBase_77A0E4A7 :
STRUCT
	{attribute addProperty Name "Device"}
	Device : Device_6E257577;
	{attribute addProperty Name "Device_Safety"}
	Device_Safety : Device_Safety_C21945A1;
	{attribute addProperty Name "Ch_A"}
	Ch_A : Ch_A_D18C6F16;
	{attribute addProperty Name "WcState"}
	WcState : WcState_B516A264;
	{attribute addProperty Name "InfoData"}
	InfoData : InfoData_358A59CF;
END_STRUCT
END_TYPE
